// TIA Portal V19 export
VAR_GLOBAL   // PLC tag table "driver"
   "Start Button 0" AT %I0.0 : Bool;
   "Stop Button 0" AT %I0.1 : Bool;
   "Selector 0 (State 0)" AT %I0.2 : Bool;
   "jog left" AT %I0.3 : Bool;
   "jog right" AT %I0.4 : Bool;
   "Potentiometer 0 (V)" AT %IW100 : Int;
   "Belt Conveyor (6m) 0 (V)" AT %QW100 : Int;
   "mem-edge1" AT %M0.0 : Bool;
   "mem-edge2" AT %M0.1 : Bool;
   "mem-edge3" AT %M0.2 : Bool;
   "mem-edge4" AT %M0.3 : Bool;
   "mem-edge5" AT %M0.4 : Bool;
   "memory-start" AT %M1.0 : Bool;
   "memory-stop" AT %M1.1 : Bool;
   "memory-3" AT %M1.2 : Bool;
   "memory-4" AT %M1.3 : Bool;
   "memory-5" AT %M1.4 : Bool;
   "mem-out scale" AT %MD100 : Real;
   "mem-val" AT %MW20 : Int;
   "mem-out norm" AT %MD104 : Real;
   "mem-jog-left" AT %MD108 : Real;
   "mem-jog-right" AT %MD112 : Real;
   spead AT %MD116 : Real;
   spead_enter AT %MD120 : Real;
END_VAR
